{attribute 'strict'}
TYPE CPICKANDPLACE :
(
	PICKANDPLACE_ESPERA,
	PICKANDPLACE_DETECCION,
	PICKANDPLACE_AGARRE,
	PICKANDPLACE_GIRO,
	PICKANDPLACE_COLOCACION,
	PICKANDPLACE_DESCENSO,
	PICKANDPLACE_LLENADO,
	PICKANDPLACE_ORIGEN
);
END_TYPE

(* stored: Version 1.1.0.1, ProductVersion 3.1.4024.12
   DUT CPICKANDPLACE: Id {edd032cf-3527-4623-a288-b28d6ca81d2a} *)
